/// this is my first test fb
/// some more doc
FUNCTION_BLOCK fb_test
VAR_INPUT
END_VAR
VAR_OUTPUT
	o_ui_countValue		:UINT;
END_VAR
VAR
END_VAR

METHOD Count : BOOL
VAR_INPUT
	i_ui_countCalue			:uint;
END_VAR
o_ui_countValue:=o_ui_countValue+i_ui_countCalue;
END_METHOD

END_FUNCTION_BLOCK

(* stored: Version 1.1.0.1
   POU fb_test: Id {95168636-7326-4d1d-a9b7-882ec4c6c6b2}, SpecialFunc None
   Method Count: Id {bee2aedd-a9a7-45cc-b84c-4d49be49a7f1} *)
